TYPE SuctionPad :
STRUCT
	enable AT %Q* : BOOL;
	occupied AT %I* : BOOL;
END_STRUCT
END_TYPE

(* stored: Version 1.1.0.1, ProductVersion 3.1.4024.11
   DUT SuctionPad: Id {2d9164d1-52b7-4c2d-9234-7506fe108a30} *)
